FUNCTION HYST (* Hystereses function *)
  (* Standard: 61499-1 *)
  (* Version 1.0, 2025-12-21, Franz Höpfinger *)
  PACKAGE OSCAT::Basic::POUs::Engineering::Control;
  IMPORT eclipse4diac::core::TypeHash;
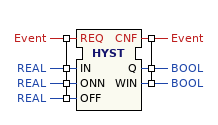
  EVENT_INPUT
    REQ WITH IN, ONN, OFF;
  END_EVENT
  EVENT_OUTPUT
    CNF WITH Q, WIN;
  END_EVENT
  VAR_INPUT
    IN : REAL;
    ONN : REAL;
    OFF : REAL;
  END_VAR
  VAR_OUTPUT
    Q : BOOL;
    WIN : BOOL;
  END_VAR
  BODY IN ST:
PACKAGE OSCAT::Basic::POUs::Engineering::Control;

(* Hystereses function *)
FUNCTION HYST
VAR_INPUT
	IN : REAL;
	ONN : REAL;
	OFF : REAL;
END_VAR

VAR_OUTPUT
	Q : BOOL;
	WIN : BOOL;
END_VAR

(*
 * version 1.0	2. jun. 2008 programmer 	hugo tested BY	oscat
 * *
 * This Hystereses function has two modes:
 * 1. if on > off then Q will be switched high when in > on and switched low when in < off.
 * 2. if on < off then Q will be switched high when in < on and switched low when in > off.
 * the output win will be high when in is between low and high.
 *)
IF ONN >= OFF THEN
	IF IN < OFF THEN
		Q := FALSE;
		WIN := FALSE;
	ELSIF  IN > ONN THEN
		Q := TRUE;
		WIN := FALSE;
	ELSE
		WIN := TRUE;
	END_IF;
ELSE
	IF IN > OFF THEN
		Q := FALSE;
		WIN := FALSE;
	ELSIF  IN < ONN THEN
		Q := TRUE;
		WIN := FALSE;
	ELSE
		WIN := TRUE;
	END_IF;
END_IF;

END_FUNCTION
(*
 * revision history hm		2.  jun 2008	rev 1.0 original version
 * *
 *)
  END_BODY
END_FUNCTION
